// SIMATIC S7-200 project (STEP 7-Micro/WIN), CPU 221 REL 01.10

SYMBOL_TABLE USER1
S1               I0.0     // NHAN CHAY
S2               I0.1     // NHAN DUNG
K                Q0.0
K3               Q0.1
K2               Q0.2
K1               Q0.3
END_SYMBOL_TABLE

ORGANIZATION_BLOCK MAIN:OB1
TITLE=PROGRAM COMMENTS
BEGIN
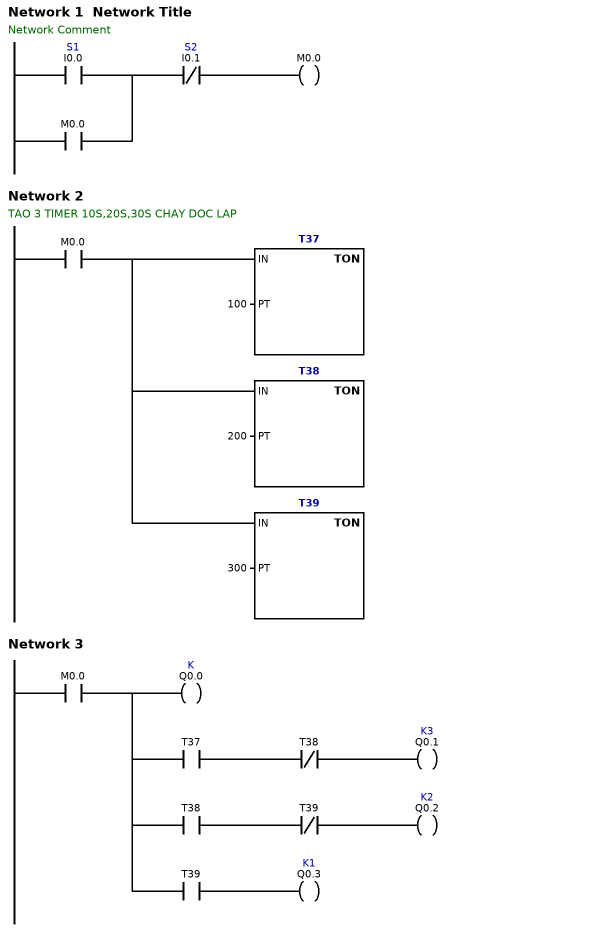
Network 1 // Network Title
// Network Comment
LD     S1:I0.0
O      M0.0
AN     S2:I0.1
=      M0.0
Network 2
// TAO 3 TIMER 10S,20S,30S CHAY DOC LAP
LD     M0.0
TON    T37, 100
TON    T38, 200
TON    T39, 300
Network 3
LD     M0.0
LPS
=      K:Q0.0
A      T37
AN     T38
=      K3:Q0.1
LRD
A      T38
AN     T39
=      K2:Q0.2
LPP
A      T39
=      K1:Q0.3
END_ORGANIZATION_BLOCK
